// TIA Portal V16 export
// export: Created 2022-03-28T07:44:09.0704204Z, ExportSetting WithDefaults, DisplayName Totally Integrated Automation Portal, DisplayVersion V16 Update 5, DisplayName TIA Portal Version Control Interface, DisplayVersion V16 Update 2, DisplayName TIA Portal Openness, DisplayVersion V16 Update 5, DisplayName STEP 7 Professional, DisplayVersion V16 Update 5, DisplayName STEP 7 Safety, DisplayVersion V16, DisplayName WinCC Professional, DisplayVersion V16 Update 5
TYPE "udtStep"
// stored: IsFailsafeCompliant false
   STRUCT
      iAction : Int;
      iPG : Int;
      iLamp : Int;
   END_STRUCT;
END_TYPE
